{attribute 'hide_all_locals'}
FUNCTION_BLOCK PUBLIC FB_ContractEmployee_1 IMPLEMENTS I_Employee
VAR_INPUT
END_VAR
VAR_OUTPUT
END_VAR
VAR
	nPersonnelNumberBacking :	UINT;
	sFirstNameBacking		:	STRING;
	sLastNameBacking		:	STRING;
	
	nHourlyPayBacking		:	UINT;
	nMonthlyHoursBacking	:	UINT;
END_VAR

METHOD GetFullName : STRING
VAR_INPUT
END_VAR
GetFullName := CONCAT(CONCAT(CONCAT(CONCAT(TO_STRING(nPersonnelNumber), ': '), sFirstName), ' '), sLastName);
END_METHOD

METHOD PUBLIC GetMonthlySalary : LREAL
VAR_INPUT
END_VAR
GetMonthlySalary := nMonthlyHours * nHourlyPay;
END_METHOD

{attribute 'monitoring' := 'variable'}
PROPERTY PUBLIC nHourlyPay : UINT
GET
nHourlyPay := nHourlyPayBacking;
END_GET
SET
nHourlyPayBacking := nHourlyPay;
END_SET
END_PROPERTY

{attribute 'monitoring' := 'variable'}
PROPERTY PUBLIC nMonthlyHours : UINT
GET
nMonthlyHours := nMonthlyHoursBacking;
END_GET
SET
nMonthlyHoursBacking := nMonthlyHours;
END_SET
END_PROPERTY

{attribute 'monitoring' := 'variable'}
PROPERTY nPersonnelNumber : UINT
GET
nPersonnelNumber := nPersonnelNumberBacking;
END_GET
SET
nPersonnelNumberBacking := nPersonnelNumber;
END_SET
END_PROPERTY

{attribute 'monitoring' := 'variable'}
PROPERTY sFirstName : STRING
GET
sFirstName := sFirstNameBacking;
END_GET
SET
sFirstNameBacking := sFirstName;
END_SET
END_PROPERTY

{attribute 'monitoring' := 'variable'}
PROPERTY sLastName : STRING
GET
sLastName := sLastNameBacking;
END_GET
SET
sLastNameBacking := sLastName;
END_SET
END_PROPERTY

END_FUNCTION_BLOCK

(* stored: Version 1.1.0.1, ProductVersion 3.1.4024.12
   POU FB_ContractEmployee_1: Id {9e3681b7-c4fc-4016-b0d2-f341b5d9712f}, SpecialFunc None
   Method GetFullName: Id {cc795efd-4dd6-47bc-89c7-c68eed1ba0c8}
   Method GetMonthlySalary: Id {b0418ec6-32f6-434c-b7b1-9fe79c7ddbb1}
   Property nHourlyPay: Id {9a08e807-5a7e-4cc6-9e9a-2a4fb57ee42e}
   Get Get: Id {772905fa-6a2d-4044-ba9b-9e84c6583352}
   Set Set: Id {435f869f-c2ee-40e5-a27f-86649047bdef}
   Property nMonthlyHours: Id {cd726a81-6e77-450e-9cf6-335e843fae94}
   Get Get: Id {78f6c95b-0f59-4865-89be-0ee3ca6020a5}
   Set Set: Id {96d6d7d0-6327-44f3-ab00-bf40abaa3c3b}
   Property nPersonnelNumber: Id {e7e31169-b080-46c8-b1cf-bcb684ad3487}
   Get Get: Id {e4a252b4-f92c-4c02-8b0f-9917ca55783e}
   Set Set: Id {360363af-2986-415a-a480-6ae3f211589d}
   Property sFirstName: Id {107316b9-4249-46a8-abe2-f3c3cc9375e0}
   Get Get: Id {0ab7f2d3-2749-484c-8b7b-221a39346aa5}
   Set Set: Id {927f5c9f-9cfc-4646-b902-1631d3642cb7}
   Property sLastName: Id {173ba9ab-37c2-45f6-b9bc-1bb61cd0aead}
   Get Get: Id {9745f6c2-f892-47d8-9a8f-4f9f1a66faba}
   Set Set: Id {51ad1137-ebf4-4fed-845c-31297a91b1a7} *)
